FUNCTION_BLOCK Test
VAR_INPUT
END_VAR
VAR_OUTPUT
END_VAR
VAR
	i,j,k : INT;
END_VAR

END_FUNCTION_BLOCK

(* stored: Version 1.1.0.1, ProductVersion 3.1.4024.2
   POU Test: Id {7dccdeb8-e15e-42f2-a785-a226f40a2e5e}, SpecialFunc None *)
